// writes traces into files, deletes too old files and monitors hdd usage
{attribute 'monitoring' := 'call'}
INTERFACE PUBLIC I_TraceHandler

// clears the internal fifo (all unwritten traces will be lost)
METHOD PUBLIC Clear

(********************************************************************************************************************************)
VAR_INPUT
END_VAR
END_METHOD

// HI = writing/deleting enabled
{attribute 'monitoring' := 'call'}
PROPERTY PUBLIC Enable : BOOL
GET
END_GET
SET
END_SET
END_PROPERTY

// folder to work within, folder must exist! (will only take effect when enabled is low)
{attribute 'monitoring' := 'call'}
PROPERTY PUBLIC Folder : A_TracePath
GET
END_GET
SET
END_SET
END_PROPERTY

// maximum file size in kilobytes
{attribute 'monitoring' := 'call'}
PROPERTY PUBLIC MaxFileSizeKB : WORD
GET
END_GET
SET
END_SET
END_PROPERTY

// HI = file is currently open
{attribute 'monitoring' := 'call'}
PROPERTY PUBLIC Opened : BOOL
GET
END_GET
END_PROPERTY

// puts a new trace line into the current file
METHOD PUBLIC Put

(********************************************************************************************************************************)
VAR_INPUT
  MsgType               : E_DebugMsgType                   := E_DebugMsgType.ERROR;
  Instance              : POINTER TO BYTE                  := 0;     // pointer to string
  Text                  : POINTER TO BYTE                  := 0;     // pointer to string
END_VAR
END_METHOD

// diagnosis & statisticals
{attribute 'monitoring' := 'call'}
PROPERTY PUBLIC Statistics : I_TraceHandlerStatistics
GET
END_GET
END_PROPERTY

END_INTERFACE

(* stored: Version 1.1.0.1, ProductVersion 3.1.4024.4
   Itf I_TraceHandler: Id {b4ff2dc4-3fe3-4d08-a8e4-9c56ceab3301}
   Folder Methods: Id {d002a3c9-a350-4c3b-8432-c1d3c5210c34}
   Folder Properties: Id {64c2a857-af1d-4dbc-a81b-62b2111136cd}
   Method Clear: Id {daf26ceb-8c50-42ea-b8e8-105cd7af90ee}
   Property Enable: Id {a54fdc2c-6c3c-4884-b4b0-9873e002d3b8}
   Get Get: Id {75b888e8-1f17-4a26-bf3f-238875824eb5}
   Set Set: Id {2bbc36a8-8eef-411d-9902-ce3d73b454ed}
   Property Folder: Id {5d75d09c-2d72-4d27-92e3-906cbd171e18}
   Get Get: Id {1ed87ea9-945e-4027-8a3b-5eec681f7033}
   Set Set: Id {44abb707-0827-4783-b9f9-4ae4aa1ab21b}
   Property MaxFileSizeKB: Id {303e1984-e23b-4307-bfaf-84bc27c4aa42}
   Get Get: Id {69567ee4-7396-473f-9586-07408b3952c7}
   Set Set: Id {231399ca-d193-40ba-92d6-9ffd52253440}
   Property Opened: Id {27c6008f-1d0b-47e6-997e-f5993c6e26ab}
   Get Get: Id {4d573152-297d-41ef-9d8c-5ec8dd1c8c3e}
   Method Put: Id {ca9e73bc-aa0a-4747-8e0c-e5540037d2cb}
   Property Statistics: Id {2c17eb65-3635-4543-83e0-e797c720bc07}
   Get Get: Id {a42e7929-f967-4613-8939-bfbc5d71e376} *)
